(* PLC project suction_head, Dassault Systèmes ControlBuild 2024x *)
(* stored: creationDateTime 2023-10-03T11:12:54-01:00 *)

(* This module simulates the behaviour of a suction head. *)
FUNCTION_BLOCK equipment_library.suction_head
  VAR_INPUT
    incPositionX : REAL := 0.0;
    incPositionY : REAL := 0.0;
    incPositionZ : REAL := 0.0;
  END_VAR
  VAR_INPUT
    vacuum : BOOL := false;
  END_VAR
  VAR_OUTPUT
    presence : BOOL := false;
  END_VAR
  VAR
    status_act_prod : DINT := 0;
    m11 : REAL := 1.0;
    m12 : REAL := 0.0;
    m13 : REAL := 0.0;
    m14 : REAL := 0.0;
    m21 : REAL := 0.0;
    m22 : REAL := 1.0;
    m23 : REAL := 0.0;
    m24 : REAL := 0.0;
    m31 : REAL := 0.0;
    m32 : REAL := 0.0;
    m33 : REAL := 1.0;
    m34 : REAL := 0.0;
    m41 : REAL := 0.0;
    m42 : REAL := 0.0;
    m43 : REAL := 0.0;
    m44 : REAL := 1.0;
    productPresence : BOOL := false;
    suckProduct : BOOL := false;
    incrementPositionX : REAL := 0.0;
    incrementPositionY : REAL := 0.0;
    incrementPositionZ : REAL := 0.0;
  END_VAR
  VAR CONSTANT
    presenceLogic : BOOL := true;
  END_VAR
  VAR
    d_presence : BOOL := false;
    v_d_presence : BOOL := false;
  END_VAR


ACTION C_source_code:
/* ----------------------------------------------------------------	*/
/* Type : Model of Operative Behaviour					*/
/* Category :  Actors and Products						*/
/* Author : Dassault Systemes						*/
/* Update date : June 2018							*/
/* ----------------------------------------------------------------	*/
/* This module simulates the behaviour of a suction head.		*/
/* ----------------------------------------------------------------	*/

/* ----------------------------------------------------------------	*/
/* Shif the suction head							*/
/* ----------------------------------------------------------------	*/
if (incPositionX != 0.0) moveXBy(myself, incPositionX);
if (incPositionY != 0.0) moveYBy(myself, incPositionY);
if (incPositionZ != 0.0) moveZBy(myself, incPositionZ);


/* ----------------------------------------------------------------	*/
/* Presence sensor								*/
/* ----------------------------------------------------------------	*/
if (d_presence) presence = v_d_presence;
else
	presence=(productPresence ^ ! presenceLogic);


/* ----------------------------------------------------------------	*/
/* Exchange informations with products				 	*/
/* ----------------------------------------------------------------	*/

suckProduct=vacuum;
productPresence=0;

/* => shift informations	*/
incrementPositionX=incPositionX;
incrementPositionY=incPositionY;
incrementPositionZ=incPositionZ;
END_ACTION
END_FUNCTION_BLOCK
